FUNCTION_BLOCK FB_StringTrimmer
VAR_INPUT
TriggerSequence : BOOL;
TrimLeft    : INT;
TrimRight   : INT;
STR         : STRING;    
END_VAR
VAR_OUTPUT
sString     : STRING;    
END_VAR
VAR    
Execute             : BOOL;
rExecuteTrig        : R_TRIG;
nStringLength       : INT;  
nStringTrimPosition : INT;
sLeftTrimmedString  : STRING; 
eStringTrim : (GET_LENGTH,TRIM_LEFT,TRIM_RIGHT,COMPLETE) := GET_LENGTH;
END_VAR

rExecuteTrig(CLK:=TriggerSequence);

IF rExecuteTrig.Q THEN
   Execute:=TRUE; 
END_IF

CASE eStringTrim OF

GET_LENGTH:
    IF Execute THEN
        nStringLength := LEN(STR);
        IF nStringLength <> 0 THEN
        eStringTrim := TRIM_LEFT;
        END_IF
     END_IF
TRIM_LEFT:
    sLeftTrimmedString:=DELETE(STR,TrimLeft,0,);
    eStringTrim := TRIM_RIGHT;
TRIM_RIGHT:
    nStringTrimPosition := nStringLength - TrimRight;      
    sString:=DELETE(sLeftTrimmedString,TrimRight,nStringTrimPosition,);
    eStringTrim := GET_LENGTH;
    Execute:=FALSE;
END_CASE

END_FUNCTION_BLOCK

(* stored: Version 1.1.0.1, ProductVersion 3.1.4024.9
   POU FB_StringTrimmer: Id {6d1403dd-cca8-4e1b-95c6-7e6876f89753}, SpecialFunc None *)
